(* PLC project Untitled1, Eclipse Foundation CIF to Structured Text 0.0 *)
(* stored: creationDateTime 1970-01-01T00:00:00Z *)

TYPE g_E : (g_LIT1, g_LIT2);
END_TYPE

TYPE TupleStruct : STRUCT
  field1 : LREAL;
  field2 : LREAL;
END_STRUCT;
END_TYPE

TYPE TupleStruct_1 : STRUCT
  field1 : TupleStruct;
  field2 : LREAL;
END_STRUCT;
END_TYPE

TYPE TupleStruct_2 : STRUCT
  field1 : DINT;
  field2 : DINT;
END_STRUCT;
END_TYPE

TYPE p_location : (p_l1, p_l6, p_l7, p_l8, p_l9, p_l10, p_l11, p_l12, p_l13, p_l14, p_l15, p_l16);
END_TYPE

PROGRAM MAIN
  VAR
    g_inp : DINT;
    p_b : BOOL;
    p_x : DINT;
    p_y : LREAL;
    p_ve : g_E;
    p_v1 : DINT;
    p_v2 : TupleStruct;
    p_v3 : TupleStruct_1;
    p_tv : TupleStruct_2;
    p_j : DINT;
    p_r : LREAL;
    p_t : LREAL;
    preset_p_t : TIME;
    p : p_location;
    firstRun : BOOL := TRUE;
  END_VAR
  VAR_TEMP
    curValue : LREAL;
    current_p : p_location;
    current_p_b : BOOL;
    current_p_j : DINT;
    current_p_r : LREAL;
    current_p_tv : TupleStruct_2;
    current_p_v3 : TupleStruct_1;
    current_p_ve : g_E;
    current_p_x : DINT;
    edge_p_1 : DINT;
    eventEnabled : BOOL;
    isProgress : BOOL;
    litStruct : TupleStruct;
    litStruct_1 : TupleStruct_1;
    litStruct_2 : TupleStruct_2;
    rightValue : TupleStruct_2;
    timeOut : BOOL;
  END_VAR

            (* Header text file for:
 *  -> (-*-) CIF PLC code generator.
 *)

(*------------------------------------------------------
 * Model overview:
 *
 * Group "g":
 * - Input variable "g.inp".
 *
 * Automaton "p":
 * - Current location of automaton "p".
 * - Discrete variable "p.b".
 * - Discrete variable "p.j".
 * - Discrete variable "p.r".
 * - Continuous variable "p.t".
 * - Discrete variable "p.tv".
 * - Discrete variable "p.v1".
 * - Discrete variable "p.v2".
 * - Discrete variable "p.v3".
 * - Discrete variable "p.ve".
 * - Discrete variable "p.x".
 * - Discrete variable "p.y".
 *
 * - PLC edge selection variable "edge_p".
 *
 * - No use of uncontrollable events.
 *
 * - Controllable event "p.evt".
 *
 *------------------------------------------------------ *)

(* --- Initialize state or update continuous variables. -------------------- *)
IF firstRun THEN
    firstRun := FALSE;

    (* Initialize the state variables. *)
    (* Initialize discrete variable "p.b". *)
    p_b := TRUE;
    (* Initialize discrete variable "p.x". *)
    p_x := 0;
    (* Initialize discrete variable "p.y". *)
    p_y := 1.23;
    (* Initialize discrete variable "p.ve". *)
    p_ve := g_LIT1;
    (* Initialize discrete variable "p.v1". *)
    p_v1 := 0;
    (* Initialize discrete variable "p.v2". *)
    litStruct.field1 := 0.0;
    litStruct.field2 := 0.0;
    p_v2 := litStruct;
    (* Initialize discrete variable "p.v3". *)
    litStruct.field1 := 0.0;
    litStruct.field2 := 0.0;
    litStruct_1.field1 := litStruct;
    litStruct_1.field2 := 0.0;
    p_v3 := litStruct_1;
    (* Initialize discrete variable "p.tv". *)
    litStruct_2.field1 := 0;
    litStruct_2.field2 := 0;
    p_tv := litStruct_2;
    (* Initialize discrete variable "p.j". *)
    p_j := 0;
    (* Initialize discrete variable "p.r". *)
    p_r := 1000000.0;
    (* Initialize continuous variable "p.t". *)
    p_t := 0.0;
    (* Reset timer of "p_t". *)
    preset_p_t := p_t;
    ton_p_t(IN := FALSE, PT := preset_p_t);
    ton_p_t(IN := TRUE, PT := preset_p_t);
    (* Initialize current location of automaton "p". *)
    p := p_l1;
ELSE
    (* Update remaining time of continuous variable "p.t". *)
    ton_p_t(IN := TRUE, PT := preset_p_t, Q => timeOut, ET => curValue);
    p_t := SEL(timeOut, preset_p_t - curValue, 0.0);
END_IF;

(* --- Process controllable events. ---------------------------------------- *)
isProgress := TRUE;
(* Perform events until none can be done anymore. *)
WHILE isProgress DO
    isProgress := FALSE;

    (*************************************************************
     * Try to perform controllable event "p.evt".
     *
     * - Automaton "p" must always synchronize.
     *************************************************************)
    eventEnabled := TRUE;
    (*******************************
     * Check each synchronizing automaton for having an edge with a true guard.
     *******************************)
    (***********
     * Test edges of automaton "p" to synchronize for event "p.evt".
     * This automaton must have an edge with a true guard to allow the event.
     *
     * Edges being tested:
     * - Location "l1":
     *   - 1st edge in the location
     * - Location "l6":
     *   - 1st edge in the location
     * - Location "l7":
     *   - 1st edge in the location
     * - Location "l8":
     *   - 1st edge in the location
     * - Location "l9":
     *   - 1st edge in the location
     * - Location "l10":
     *   - 1st edge in the location
     * - Location "l11":
     *   - 1st edge in the location
     * - Location "l12":
     *   - 1st edge in the location
     * - Location "l13":
     *   - 1st edge in the location
     * - Location "l14":
     *   - 1st edge in the location
     * - Location "l15":
     *   - 1st edge in the location
     ***********)
    IF p = p_l1 THEN
        edge_p_1 := 1;
    ELSIF p = p_l6 THEN
        edge_p_1 := 2;
    ELSIF p = p_l7 THEN
        edge_p_1 := 3;
    ELSIF p = p_l8 THEN
        edge_p_1 := 4;
    ELSIF p = p_l9 THEN
        edge_p_1 := 5;
    ELSIF p = p_l10 THEN
        edge_p_1 := 6;
    ELSIF p = p_l11 THEN
        edge_p_1 := 7;
    ELSIF p = p_l12 THEN
        edge_p_1 := 8;
    ELSIF p = p_l13 THEN
        edge_p_1 := 9;
    ELSIF p = p_l14 THEN
        edge_p_1 := 10;
    ELSIF p = p_l15 THEN
        edge_p_1 := 11;
    ELSE
        (* The automaton has no edge with a true guard. Skip to the next event. *)
        eventEnabled := FALSE;
    END_IF;
    (* All checks have been done. If variable "eventEnabled" still holds, event "p.evt" can occur. *)
    IF eventEnabled THEN
        isProgress := TRUE;
        (* Make temporary copies of assigned variables to preserve the old values while assigning new values. *)
        current_p := p;
        current_p_b := p_b;
        current_p_j := p_j;
        current_p_r := p_r;
        current_p_tv := p_tv;
        current_p_v3 := p_v3;
        current_p_ve := p_ve;
        current_p_x := p_x;
        (*******************************
         * Perform the assignments of each synchronizing automaton.
         *******************************)
        (* Perform assignments of automaton "p". *)
        IF edge_p_1 = 1 THEN
            (* Perform assignments of the 1st edge in location "p.l1". *)
            (* Perform update of discrete variable "p.tv". *)
            litStruct_2.field1 := 1;
            litStruct_2.field2 := 2;
            p_tv := litStruct_2;
            (* Perform update of current location of automaton "p". *)
            p := p_l6;
        ELSIF edge_p_1 = 2 THEN
            (* Perform assignments of the 1st edge in location "p.l6". *)
            (* Perform update of discrete variable "p.x". *)
            p_x := 3;
            (* Perform update of discrete variable "p.j". *)
            p_j := 4;
            (* Perform update of current location of automaton "p". *)
            p := p_l7;
        ELSIF edge_p_1 = 3 THEN
            (* Perform assignments of the 1st edge in location "p.l7". *)
            rightValue := current_p_tv;
            (* Perform update of discrete variable "p.x". *)
            p_x := rightValue.field1;
            (* Perform update of discrete variable "p.j". *)
            p_j := rightValue.field2;
            (* Perform update of current location of automaton "p". *)
            p := p_l8;
        ELSIF edge_p_1 = 4 THEN
            (* Perform assignments of the 1st edge in location "p.l8". *)
            (* Perform update of discrete variable "p.tv". *)
            p_tv.field1 := 5;
            (* Perform update of current location of automaton "p". *)
            p := p_l9;
        ELSIF edge_p_1 = 5 THEN
            (* Perform assignments of the 1st edge in location "p.l9". *)
            (* Perform update of discrete variable "p.tv". *)
            p_tv.field2 := 6;
            (* Perform update of discrete variable "p.j". *)
            p_j := 7;
            (* Perform update of current location of automaton "p". *)
            p := p_l10;
        ELSIF edge_p_1 = 6 THEN
            (* Perform assignments of the 1st edge in location "p.l10". *)
            (* Perform update of discrete variable "p.v3". *)
            p_v3.field1.field2 := 7.8;
            (* Perform update of current location of automaton "p". *)
            p := p_l11;
        ELSIF edge_p_1 = 7 THEN
            (* Perform assignments of the 1st edge in location "p.l11". *)
            (* Perform update of discrete variable "p.v3". *)
            litStruct.field1 := 1.2;
            litStruct.field2 := 3.4;
            litStruct_1.field1 := litStruct;
            litStruct_1.field2 := 5.6;
            p_v3 := litStruct_1;
            (* Perform update of current location of automaton "p". *)
            p := p_l12;
        ELSIF edge_p_1 = 8 THEN
            (* Perform assignments of the 1st edge in location "p.l12". *)
            (* Perform update of discrete variable "p.j". *)
            p_j := current_p_j + 1;
            (* Perform update of current location of automaton "p". *)
            p := p_l13;
        ELSIF edge_p_1 = 9 THEN
            (* Perform assignments of the 1st edge in location "p.l13". *)
            (* Perform update of discrete variable "p.b". *)
            p_b := FALSE;
            (* Perform update of current location of automaton "p". *)
            p := p_l14;
        ELSIF edge_p_1 = 10 THEN
            (* Perform assignments of the 1st edge in location "p.l14". *)
            IF NOT current_p_b THEN
                (* Perform update of discrete variable "p.ve". *)
                p_ve := g_LIT2;
            END_IF;
            (* Perform update of current location of automaton "p". *)
            p := p_l15;
        ELSIF edge_p_1 = 11 THEN
            (* Perform assignments of the 1st edge in location "p.l15". *)
            (* Perform update of discrete variable "p.r". *)
            p_r := DINT_TO_LREAL(g_inp) + 10.0;
            (* Perform update of current location of automaton "p". *)
            p := p_l16;
        END_IF;
    END_IF;
END_WHILE;
          
END_PROGRAM

CONFIGURATION Untitled1
  RESOURCE Untitled1 ON PLC
    VAR_GLOBAL  (* TIMERS *)
      ton_p_t : TON;
    END_VAR
    TASK PlcTask(INTERVAL := T#10ms, PRIORITY := 20);
    PROGRAM MAIN WITH PlcTask : MAIN;
  END_RESOURCE
END_CONFIGURATION
